Fanuc KAREL source: NC0080.KL

PROGRAM NC0080
%NOLOCKGROUP
ROUTINE R
VAR
S1:INTEGER
BEGIN
S1=1
WHILE (S1<2) DO
WHILE (S1<2) DO
WHILE (S1<2) DO
WHILE (S1<2) DO
WHILE (S1<2) DO
WHILE (S1<2) DO
WHILE (S1<2) DO
WHILE (S1<2) DO
WHILE (S1<2) DO
WHILE (S1<2) DO
WHILE (S1<2) DO
WHILE (S1<2) DO
WHILE (S1<2) DO
WHILE (S1<2) DO
WHILE (S1<2) DO
WHILE (S1<2) DO
WHILE (S1<2) DO
WHILE (S1<2) DO
S1=(S1+1)
ENDWHILE
ENDWHILE
ENDWHILE
ENDWHILE
ENDWHILE
ENDWHILE
ENDWHILE
ENDWHILE
ENDWHILE
ENDWHILE
ENDWHILE
ENDWHILE
ENDWHILE
ENDWHILE
ENDWHILE
ENDWHILE
ENDWHILE
ENDWHILE
END R
BEGIN
R
END NC0080
